FUNCTION_BLOCK FB_ScaleTrigger
VAR_INPUT
	scaleEntry_input : BOOL;
	
	scaleExit_input : BOOL;
END_VAR
VAR_OUTPUT
	ScaleEntryEdgeDetected : BOOL;
	
	ScaleExitEdgeDetected : BOOL;
END_VAR
VAR
	rTrigScaleEntry : Tc2_Standard.R_TRIG;
	
	fTrigScaleExit : Tc2_Standard.F_TRIG;
END_VAR

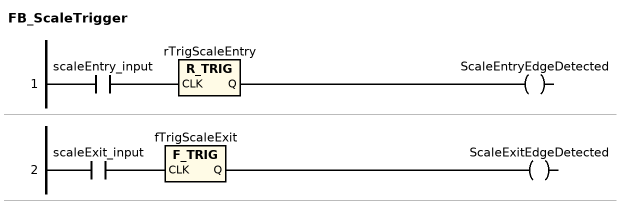
// NETWORK 1
rTrigScaleEntry(CLK := scaleEntry_input); // R_TRIG
ScaleEntryEdgeDetected := rTrigScaleEntry.Q;

// NETWORK 2
fTrigScaleExit(CLK := scaleExit_input); // F_TRIG
ScaleExitEdgeDetected := fTrigScaleExit.Q;

END_FUNCTION_BLOCK

(* stored: Version 1.1.0.1, ProductVersion 3.1.4024.13
   POU FB_ScaleTrigger: Id {509c8924-523b-4e0f-bfe7-d9051d5707bd}, SpecialFunc None *)
